TYPE Serial_COMBUFFER :
STRUCT
(**)
	(* PLC to IO interface *)
	txBuffer 		: ComBuffer;
	rxBuffer 		: ComBuffer;
(**)
(**)	
	(* Buffers for EL COM *)
	rxElComBuffer AT %I* 	: EL6inData22B;
	txElComBuffer AT %Q* 	: EL6outData22B;
(**)
(*
	(* Buffers for PC COM *)
	rxPcComBuffer AT %I* 	: PcComInData;
	txPcComBuffer AT %Q* 	: PcComOutData;
*)
END_STRUCT
END_TYPE

(* stored: Version 1.1.0.1, ProductVersion 3.1.0.36
   DUT Serial_COMBUFFER: Id {c96ffc7c-11c3-44f3-a8bd-4a56f912f985} *)
